PROGRAM Zone_Monitoring
VAR
    fbZoneMonitoring: FB_ZoneMonitoring;
END_VAR

fbZoneMonitoring(
    iSafetyProvider := Motion_Safety.fbMotionSafety,
	stSafety := Motion_Safety.stSafety,
    aErrorID =>,
    aErrorMsg =>,
    nAlarmGrpBitNumber =>);

END_PROGRAM

(* stored: Version 1.1.0.1
   POU Zone_Monitoring: Id {2b0d7b86-187f-0bc2-2f54-f64dd930b8f4}, SpecialFunc None *)
